// TwinCAT 3 PLC project Potentiometer_Inlezen_VISU
// ProgramVersion: 3.1.4024.0
// libraries:
//   Tc2_Standard, * (Beckhoff Automation GmbH)
//   Tc2_System, * (Beckhoff Automation GmbH)
//   Tc3_Module, * (Beckhoff Automation GmbH)
//   VisuDialogs, * (System)
//   VisuSymbols,3.5.10.0,System
// project tree:
//   / GlobalTextList.TcGTLO, PlcTask.TcTTO, Visualization Manager.TcVMO (not stored)
//   POUs/ MAIN.TcPOU
//   VISUs/ Visualization.TcVIS
// (motion and I/O tree: see PLC project potentiometer_inlezen)
// real-time tasks:
//   TASK PlcTask: cycle T#10ms, priority 20, ADS port 350
//   TASK PlcTask1: cycle T#10ms, priority 21, ADS port 351
//   TASK PlcTask2: cycle T#10ms, priority 22, ADS port 352
//   TASK PlcTask3: cycle T#10ms, priority 26, ADS port 353
//   TASK PlcTask4: cycle T#10ms, priority 25, ADS port 354
//   TASK PlcTask5: cycle T#10ms, priority 24, ADS port 355
//   TASK PlcTask6: cycle T#10ms, priority 23, ADS port 356
//   TASK PlcTask7: cycle T#10ms, priority 27, ADS port 357

CONFIGURATION Potentiometer_Inlezen_VISU
    RESOURCE PLC ON TwinCAT3
        TASK PlcTask(INTERVAL := T#10ms, PRIORITY := 22);
        PROGRAM MAIN WITH PlcTask : MAIN;
    END_RESOURCE
END_CONFIGURATION

// ---- POUs/MAIN.TcPOU
PROGRAM MAIN
VAR
	Waarde: BYTE;
	potentiometer: INT;
	nScaledMax: INT := 10;
END_VAR

(*
Potentiometer inlezen met visualisatie
Gebruik een visualisatie om de maximumwaarde en de output te tonen, alsook om de maximumwaarde te verschalen.
Rechtermuisklik op de folder VISU, selecteer 'add new' en vervolgens een VISUALISATION. Sleep vanuit de toolbox twee rectangles naar het canvas. 
Via properties window configureer je deze rectangles om de maximumwaarde nScaledMax te tonen en in te geven, en om de verschaalde output te tonen in de visu. 
*)

Waarde:=LREAL_TO_BYTE(nScaledMax*(potentiometer/32767.0));

END_PROGRAM

// ---- GlobalTextList.TcGTLO
TEXTLIST GlobalTextList
  387 = 'De max waarde is %d'
  898 = 'De verschaalde waarde %d'
END_TEXTLIST

// ---- VISUs/Visualization.TcVIS
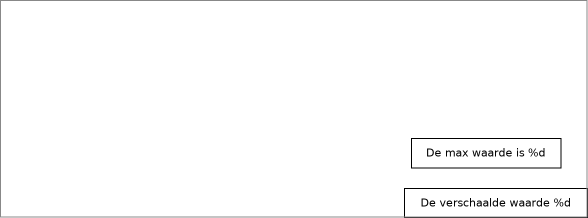
VISUALIZATION Visualization  // 588x218
    Rectangle (411,138 150x30), "De max waarde is %d", text variable: MAIN.nScaledMax
        OnMouseDown: write the text variable via Default
    Rectangle (404,188 184x30), "De verschaalde waarde %d", text variable: MAIN.Waarde
END_VISUALIZATION
